// LS Electric XG5000 project: 20240307
// PLC LSPLC
// module base 0 slot 0: 입출력 모듈:XBM-DN/DP32HP (DC 24V입력/TR 출력, 32점)
// module base 0 slot 1: 내장위치결정:XBF-PO06E (오픈컬렉터형, 6축)

PROGRAM NewProgram (task: 스캔 프로그램)

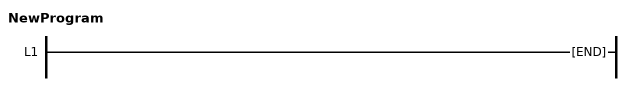
; L1
END